{attribute addProperty BoxType "BK1250-0000-0016"}
{attribute addProperty Id "Term_396_KL1002KL1002_D229A9CA00"}
{attribute addProperty CRC "1777678844"}
{attribute addProperty SizeInBites "0"}
{attribute addProperty SizeInBytes "0"}
TYPE A_0015_BK1250_0000_0016_69F539FC EXTENDS BK1250_A5F67C82 :
STRUCT
	{attribute addProperty Name "Term_396_KL1002"}
	Term_396_KL1002 : KL1002_D229A9CA;
END_STRUCT
END_TYPE

(* stored: Version 1.2.0.0, ProductVersion 3.1.4024.9
   DUT A_0015_BK1250_0000_0016_69F539FC: Id {d3d62ba5-bd72-4ad5-a7ad-f1224b70b578} *)
